# EPICS StreamDevice protocol: protocols/acq494.proto
Terminator = LF;
ExtraInput = Ignore;

# T50R_[1-4] or T50R (global) value 0 or 1
setT50R {
	out "T50R\$1 %d";
	in;
}

getT50R {
	out "T50R\$1";
	in "%d";
}

setMask {
	out "scount_evt_ch\$1 %d";
	in;
}

getMask {
	out "scount_evt_ch\$1";
	in "%d";
}
